FUNCTION_BLOCK E_D_FF
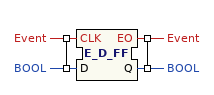
  EVENT_INPUT
    CLK WITH D;
  END_EVENT
  EVENT_OUTPUT
    EO WITH Q;
  END_EVENT
  VAR_INPUT
    D : BOOL;
  END_VAR
  VAR_OUTPUT
    Q : BOOL;
  END_VAR
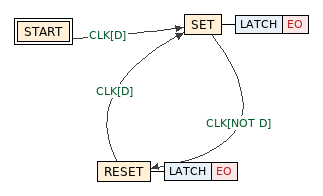
  EC_STATES
    START;
    SET : LATCH -> EO;
    RESET : LATCH -> EO;
  END_STATES
  EC_TRANSITIONS
    START TO SET := CLK[D];
    SET TO RESET := CLK[NOT D];
    RESET TO SET := CLK[D];
  END_TRANSITIONS
  ALGORITHM LATCH IN ST:
Q := D;&#38;#10;
  END_ALGORITHM
END_FUNCTION_BLOCK
